{attribute 'qualified_only'}
{attribute 'strict'}
TYPE E_CX_NVDataOpMode : (
	//E_CX_NVDATA_OPMODE_IDLE,
	//E_CX_NVDATA_OPMODE_EL6080,
	//E_CX_NVDATA_OPMODE_NOVRAM,
	//E_CX_NVDATA_OPMODE_BINARYFILE
	DUMMY
);
END_TYPE

(* stored: Version 1.1.0.1
   DUT E_CX_NVDataOpMode: Id {56fcd908-f2cc-440a-8768-3551b5a30cb3} *)
